TYPE "KukaRobot_HMI"
VERSION : 0.1
   STRUCT
      PGNO_PBIT : USInt;
      EXT_START : Bool;
      MOVE_ENABLE : Bool;
      CONF_MESS : Bool;
      DRIVES_OFF : Bool;
      DRIVES_ON : Bool;
      I_O_ACT : Bool;
      RC_RDY1 : Bool;
      ALARM_STOP : Bool;
      USER_SAF : Bool;
      PERI_RDY : Bool;
      ROB_CAL : Bool;
      I_O_ACTCONF : Bool;
      STOPMESS : Bool;
      ALARM_STOP_INTERN : Bool;
      PGNO_FBIT_REFL : USInt;
      PRO_ACT : Bool;
      APPL_RUN : Bool;
      PRO_MOVE : Bool;
      IN_HOME : Bool;
      ON_PATH : Bool;
      NEAR_POSRET : Bool;
      T1 : Bool;
      T2 : Bool;
      AUT : Bool;
      EXT : Bool;
      TaskMode : USInt;
      PartType : USInt;
      SpeedSet : USInt;
      HomeSeqStart : Bool;
      AutoCycleStart : Bool;
      CurrentMode : USInt;
      CurrentPartType : USInt;
      SpeedActual : USInt;
      ProgramSequence : USInt;
      WaitForHomeSeqStart : Bool;
      GoHomeFail : Bool;
      HomeSeqOK : Bool;
      WaitForAutoCycleStart : Bool;
      iTaskMode : USInt;
      iPartType : USInt;
      iSpeedValue : USInt;
      iPGNO : USInt;
      AutoStart : Bool;
      SrartHome : Bool;
      StartAutoCycle : Bool;
      Ready : Bool;
      StartComplete : Bool;
      StartUpTimeOut : Bool;
      Warning : Bool;
      Error : Bool;
      ErrorCode : Int;
      Seconds : Int;
      Minute : Int;
      Hours : DInt;
      CountPulse : Bool;
      StartSeq : Int;
   END_STRUCT;

END_TYPE

